FUNCTION_BLOCK OneMoreInnerBlock
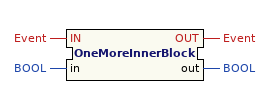
  EVENT_INPUT
    IN;
  END_EVENT
  EVENT_OUTPUT
    OUT;
  END_EVENT
  VAR_INPUT
    in : BOOL;
  END_VAR
  VAR_OUTPUT
    out : BOOL;
  END_VAR
  EC_STATES
    START;
  END_STATES
END_FUNCTION_BLOCK
